(* Logix 5000 project; controller STAT 1756-L72 rev 20.12; software revision 20.04; part 14 of 34 *)
(* tags used below, declared in another part *)
   B14 : DINT[30];
   B15 : DINT[30];
   B16 : DINT[30];
   B17 : DINT[30];
   B3 : DINT[256];
   B9 : DINT[40];
   DateTime : DINT[7];   // DINT array tag for retrieve wallclock time through GSV created during conversion
   I19_000_Bit01 : ALIAS FOR I19[0].1;   // VANNE ALIBERT FERMEE
   I19_000_Bit07 : ALIAS FOR I19[0].7;   // LACK DETECTIE H2SO4
   I19_000_Bit08 : ALIAS FOR I19[0].8;   // LACK DETECTIE NAOH
   I19_001_Bit02 : ALIAS FOR I19[1].2;
   I19_001_Bit04 : ALIAS FOR I19[1].4;
   I1_008_Bit00 : ALIAS FOR I1[8].0;   // Noodstop gedrukt
   I1_008_Bit12 : ALIAS FOR I1[8].12;   // start
   I1_009_Bit00 : ALIAS FOR I1[9].0;   // Spanning 220 V nuts ok
   I1_009_Bit01 : ALIAS FOR I1[9].1;   // Spanning 220 v ac ok
   I1_009_Bit02 : ALIAS FOR I1[9].2;   // Spanning 24 v dc ok
   I1_009_Bit03 : ALIAS FOR I1[9].3;   // Thermische storing pomp 1
   I1_009_Bit07 : ALIAS FOR I1[9].7;   // Thermische storing pomp 2
   I1_009_Bit11 : ALIAS FOR I1[9].11;   // Thermische storing pomp 3
   I1_009_Bit15 : ALIAS FOR I1[9].15;   // Thermische storing pomp pd1 ok
   I1_010_Bit00 : ALIAS FOR I1[10].0;   // PD1 spanning ok op regelaar
   I1_010_Bit02 : ALIAS FOR I1[10].2;   // Thermische storng pomp pd2 ok
   I1_010_Bit03 : ALIAS FOR I1[10].3;   // PD2 spanning ok op regelaar
   I1_010_Bit05 : ALIAS FOR I1[10].5;   // Vlotterschak lal stormbekken
   I1_010_Bit06 : ALIAS FOR I1[10].6;   // Storing voeding promag 33
   I1_010_Bit08 : ALIAS FOR I1[10].8;   // Fout promag 33
   I1_010_Bit10 : ALIAS FOR I1[10].10;   // Noodstop relais ok stormbekken
   I1_016_Bit00 : ALIAS FOR I1[16].0;   // CL2 noodstop gedrukt
   I1_016_Bit10 : ALIAS FOR I1[16].10;   // conduc 3 alarm
   I1_016_Bit13 : ALIAS FOR I1[16].13;   // Niveau lus5 kontakt3
   I1_017_Bit00 : ALIAS FOR I1[17].0;   // CL3 noodstop gedrukt
   I1_017_Bit10 : ALIAS FOR I1[17].10;   // conduc 4 alarm
   I1_017_Bit13 : ALIAS FOR I1[17].13;   // Niveau lus6 kontakt3
   I1_017_Bit14 : ALIAS FOR I1[17].14;   // Niveau A3 vlotter niveau
   I1_018_Bit00 : ALIAS FOR I1[18].0;   // CL4 noodstop gedrukt
   I1_018_Bit10 : ALIAS FOR I1[18].10;   // conduc 5 alarm
   I1_018_Bit13 : ALIAS FOR I1[18].13;   // Niveau lus7 kontakt3
   I1_019_Bit00 : ALIAS FOR I1[19].0;   // 220V ok aan lijn 123
   I2_000_Bit00 : ALIAS FOR I2[0].0;   // Deelnoodstop cl2 lijn 1
   I2_000_Bit01 : ALIAS FOR I2[0].1;   // Deelnoodstop cl3 lijn 3
   I2_000_Bit02 : ALIAS FOR I2[0].2;   // Deelnoodstop cl4
   I2_000_Bit03 : ALIAS FOR I2[0].3;   // Deelnoodstop cl5 lijn 4
   I2_000_Bit04 : ALIAS FOR I2[0].4;   // Deelnoodstop cl6 eurowater
   I2_000_Bit05 : ALIAS FOR I2[0].5;   // Deelnoodstop cl7 IBT A
   I2_000_Bit06 : ALIAS FOR I2[0].6;   // Deelnoodstop cl7 IBT B
   I2_000_Bit07 : ALIAS FOR I2[0].7;   // Deelnoodstop cl7 IBT C
   I2_000_Bit08 : ALIAS FOR I2[0].8;   // Voeidng 220V ok
   I2_000_Bit09 : ALIAS FOR I2[0].9;   // Storing voeding lijn 1 cl 2
   I2_000_Bit10 : ALIAS FOR I2[0].10;   // Storing voeding lijn 2 cl 3
   I2_000_Bit11 : ALIAS FOR I2[0].11;   // Storing voeding lijn 3 cl 4
   I2_000_Bit12 : ALIAS FOR I2[0].12;   // Storing voeding lijn 4 cl 5
   I2_000_Bit13 : ALIAS FOR I2[0].13;   // Storing voeding lijn deel eurowater cl 6
   I2_000_Bit14 : ALIAS FOR I2[0].14;   // Storing voedingslijn IBT-A CL 7
   I2_000_Bit15 : ALIAS FOR I2[0].15;   // Storing voedingslijn IBT-B CL 8
   I2_001_Bit00 : ALIAS FOR I2[1].0;   // Storing voedingslijn IBT-C CL 9
   I2_001_Bit01 : ALIAS FOR I2[1].1;   // Voeding meting 220V ok
   I2_001_Bit02 : ALIAS FOR I2[1].2;   // Voeding DC 24 ok
   I2_001_Bit03 : ALIAS FOR I2[1].3;   // Storing voeding 24V DC algemeen
   I2_001_Bit04 : ALIAS FOR I2[1].4;   // Storing voeding 24V ingangen
   I2_001_Bit05 : ALIAS FOR I2[1].5;   // Storing 24V meting
   I2_001_Bit06 : ALIAS FOR I2[1].6;   // Voeding uitgang 24V
   I2_001_Bit08 : ALIAS FOR I2[1].8;   // Motor p11 lijn1 thermische storing
   I2_001_Bit10 : ALIAS FOR I2[1].10;   // Motor p12 lijn1 thermische storing
   I2_001_Bit12 : ALIAS FOR I2[1].12;   // Motor p13 lijn2 thermische storing
   I2_001_Bit14 : ALIAS FOR I2[1].14;   // Motor p14 lijn2 thermische storing
   I3_000_Bit00 : ALIAS FOR I3[0].0;   // Motor p15 lijn3 thermische storing
   I3_000_Bit02 : ALIAS FOR I3[0].2;   // Motor p16 lijn3 thermische storing
   I3_000_Bit04 : ALIAS FOR I3[0].4;   // Motor p17 lijn4 thermische storing
   I3_000_Bit06 : ALIAS FOR I3[0].6;   // Motor p18 lijn4 thermische storing
   I3_000_Bit07 : ALIAS FOR I3[0].7;   // Motor pro 1 voedingpomp osmose 1 Thermische storing
   I3_000_Bit09 : ALIAS FOR I3[0].9;   // Motor pro 1 voedingpomp osmose 1 in driehoek
   I3_000_Bit11 : ALIAS FOR I3[0].11;   // Motor pro2 voedingpomp osmose 2 Thermische storing
   I3_000_Bit13 : ALIAS FOR I3[0].13;   // Motor pro 2 voedingpomp osmose 2 in driehoek
   I3_000_Bit15 : ALIAS FOR I3[0].15;   // Motor P21 Thermische storing Kuip AZ
   I3_001_Bit03 : ALIAS FOR I3[1].3;   // Thermische storing motor P22 kuip AZ
   I3_001_Bit07 : ALIAS FOR I3[1].7;   // Thermische storing motor PRO3 voedingsp. osmose 3
   I3_001_Bit09 : ALIAS FOR I3[1].9;   // Motor voedingspomp osmose 3 in drie
   I3_001_Bit11 : ALIAS FOR I3[1].11;   // Motor P21 reinigingspomp membraam
   I3_001_Bit13 : ALIAS FOR I3[1].13;   // Thermische storing S2 ventilator
   I3_001_Bit15 : ALIAS FOR I3[1].15;   // Thermische storing voedingspomp fabriek 1
   I4_000_Bit03 : ALIAS FOR I4[0].3;   // Thermische storing voedingspomp fabriek 2
   I4_000_Bit08 : ALIAS FOR I4[0].8;   // Thermische storing motor p 5 ok
   I4_000_Bit10 : ALIAS FOR I4[0].10;   // Thermische storing p6 ok
   I4_000_Bit15 : ALIAS FOR I4[0].15;   // thermische storing frequentieregelaar motor p25
   I4_001_Bit01 : ALIAS FOR I4[1].1;   // Thermische storing freqreg p20
   I4_001_Bit03 : ALIAS FOR I4[1].3;   // Motor AG1 mixer vat neutral thermische st ok
   I4_001_Bit05 : ALIAS FOR I4[1].5;   // Motor acide thermische st ok
   I4_001_Bit07 : ALIAS FOR I4[1].7;   // Motor acide 4 thermische st ok
   I4_001_Bit09 : ALIAS FOR I4[1].9;   // Motor soude 5 thermische st ok
   I4_001_Bit11 : ALIAS FOR I4[1].11;   // Motor soude 6 thermische st ok
   I4_001_Bit13 : ALIAS FOR I4[1].13;   // Motor ag2 mixer thermische st ok
   I4_001_Bit15 : ALIAS FOR I4[1].15;   // Motor ag3 mixer thermische st ok
   I5_000_Bit00 : ALIAS FOR I5[0].0;   // thermische storing motor doseerpop1 pd7
   I5_000_Bit01 : ALIAS FOR I5[0].1;   // spanning op motor freqreg doseer floculaat
   I5_000_Bit02 : ALIAS FOR I5[0].2;   // storing freqreg doseer floculaat
   I5_000_Bit03 : ALIAS FOR I5[0].3;   // thermische storing motor freqreg doseer floculaat pd8
   I5_000_Bit04 : ALIAS FOR I5[0].4;   // spanning op motor freqreg doseer floculaat pd8
   I5_000_Bit05 : ALIAS FOR I5[0].5;   // storing freqreg doseer floculaat pd8
   I5_000_Bit07 : ALIAS FOR I5[0].7;   // thermische storing motor zuiveringspomp p19
   I5_000_Bit09 : ALIAS FOR I5[0].9;   // thermische storing motor zuiveringspomp p19b
   I5_000_Bit10 : ALIAS FOR I5[0].10;   // thermische storing motor PM1
   I5_000_Bit11 : ALIAS FOR I5[0].11;   // spanning op motor freqreg recerculatiep. dec. ingang 1
   I5_000_Bit12 : ALIAS FOR I5[0].12;   // fout freqreg recerculatiep. dec. ingang 1
   I5_000_Bit13 : ALIAS FOR I5[0].13;   // thermische storing motor recirculatiep. dec. ingang 2
   I5_000_Bit14 : ALIAS FOR I5[0].14;   // spanning freqreg. recirculatiep. dec. ingang 2
   I5_000_Bit15 : ALIAS FOR I5[0].15;   // fout freqreg recerculatiep. dec. ingang 2
   I5_001_Bit00 : ALIAS FOR I5[1].0;   // thermische storing motor evacuatiepomp dec. ingang 1
   I5_001_Bit01 : ALIAS FOR I5[1].1;   // spanning freqreg. evacuatiepomp decanter ingang 1
   I5_001_Bit02 : ALIAS FOR I5[1].2;   // fout freqreg pm3 evacuatiep. dec. ingang 1
   I5_001_Bit03 : ALIAS FOR I5[1].3;   // thermische storing motor evacuatiepomp dec. ingang 2
   I5_001_Bit04 : ALIAS FOR I5[1].4;   // spanning freqreg. evacuatiepomp decanter ingang 2
   I5_001_Bit05 : ALIAS FOR I5[1].5;   // fout freqreg pm4 evacuatiep. dec. ingang 2
   I5_001_Bit06 : ALIAS FOR I5[1].6;   // thermische storing voedingspomp 1 osmose ok
   I5_001_Bit08 : ALIAS FOR I5[1].8;   // thermische storing voedingspomp 2 osmose ok
   I5_001_Bit10 : ALIAS FOR I5[1].10;   // thermische storing voedingspomp 3 osmose ok
   I6_000_Bit10 : ALIAS FOR I6[0].10;   // pressostaat osmose1
   I6_000_Bit11 : ALIAS FOR I6[0].11;   // pressostaat osmose2
   I6_000_Bit12 : ALIAS FOR I6[0].12;   // pressostaat osmose3
   I6_001_Bit06 : ALIAS FOR I6[1].6;   // debietsmeting q2 fout 1
   I6_001_Bit09 : ALIAS FOR I6[1].9;   // debietsmeting q3 fout 1
   I6_001_Bit11 : ALIAS FOR I6[1].11;   // Ph meting vervuild water kontakt 1
   I7_000_Bit00 : ALIAS FOR I7[0].0;   // ph meting fout gerecycleerd water
   I7_000_Bit01 : ALIAS FOR I7[0].1;   // lus2 niveau kontakt 1
   I7_000_Bit03 : ALIAS FOR I7[0].3;   // lus2 niveau kontakt 3
   I7_000_Bit04 : ALIAS FOR I7[0].4;   // lus3 niveau kontakt 1
   I7_000_Bit06 : ALIAS FOR I7[0].6;   // lus3 niveau kontakt 3
   I7_000_Bit10 : ALIAS FOR I7[0].10;   // zeer hoog alarm ketel clarifee
   I7_000_Bit13 : ALIAS FOR I7[0].13;   // zeer laag alarm ketel clarifee
   I7_001_Bit03 : ALIAS FOR I7[1].3;   // Conductiviteit 1 alarm 3
   I7_001_Bit06 : ALIAS FOR I7[1].6;   // Conductiviteit 2 kontakt alarm
   I7_001_Bit12 : ALIAS FOR I7[1].12;   // Lus 8 niveau kontakt 3
   N12 : DINT[230];
   N13 : DINT[230];
   N26 : DINT[256];
   O14_001_Bit13 : ALIAS FOR O14[1].13;   // RO1_EV2 RO1_EV2
   O15_000_Bit01 : ALIAS FOR O15[0].1;   // RO2_EV2 RO2_EV2
   O15_000_Bit05 : ALIAS FOR O15[0].5;   // RO3_EV2 RO3_EV2
   O1_011_Bit00 : ALIAS FOR O1[11].0;
   O1_011_Bit03 : ALIAS FOR O1[11].3;
   T27 : TIMER[100];
   T4 : TIMER[200];
(* ibt, continued *)

ROUTINE _17_DEF_TEL   (* ladder *)
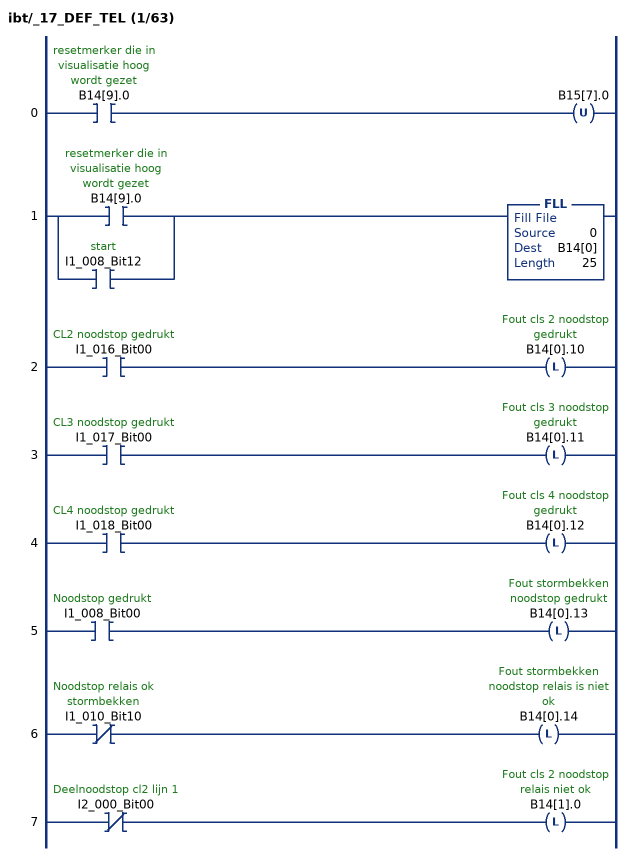
   0: XIC(B14[9].0)OTU(B15[7].0);
   1: [XIC(B14[9].0) ,XIC(I1_008_Bit12) ]FLL(0,B14[0],25);
   2: XIC(I1_016_Bit00)OTL(B14[0].10);
   3: XIC(I1_017_Bit00)OTL(B14[0].11);
   4: XIC(I1_018_Bit00)OTL(B14[0].12);
   5: XIC(I1_008_Bit00)OTL(B14[0].13);
   6: XIO(I1_010_Bit10)OTL(B14[0].14);
   7: XIO(I2_000_Bit00)OTL(B14[1].0);
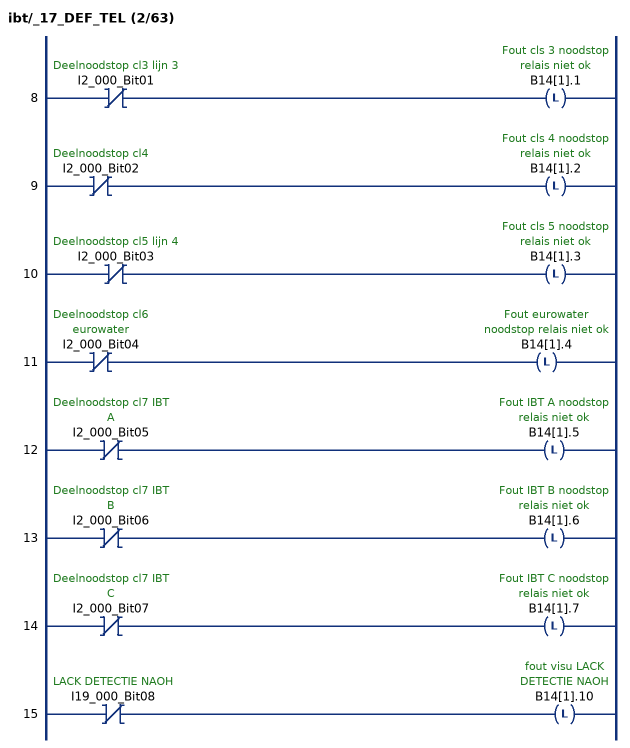
   8: XIO(I2_000_Bit01)OTL(B14[1].1);
   9: XIO(I2_000_Bit02)OTL(B14[1].2);
   10: XIO(I2_000_Bit03)OTL(B14[1].3);
   11: XIO(I2_000_Bit04)OTL(B14[1].4);
   12: XIO(I2_000_Bit05)OTL(B14[1].5);
   13: XIO(I2_000_Bit06)OTL(B14[1].6);
   14: XIO(I2_000_Bit07)OTL(B14[1].7);
   15: XIO(I19_000_Bit08)OTL(B14[1].10);
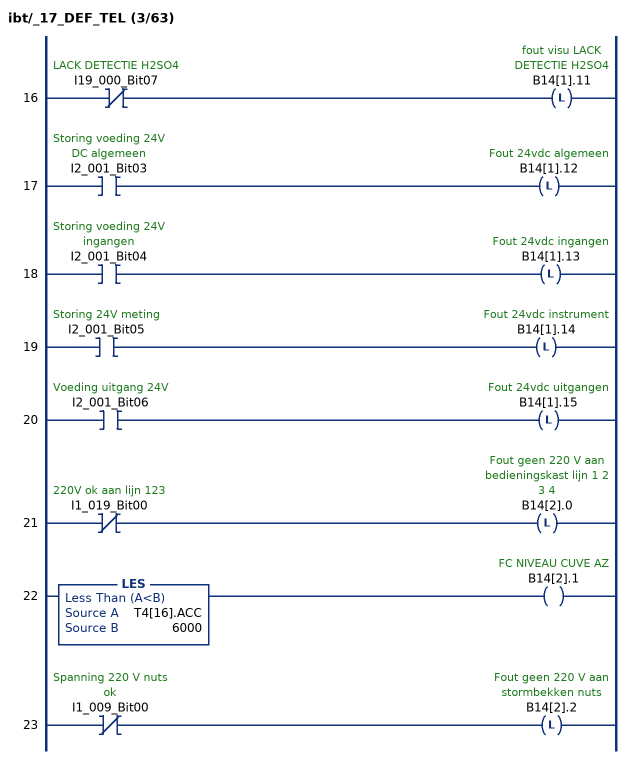
   16: XIO(I19_000_Bit07)OTL(B14[1].11);
   17: XIC(I2_001_Bit03)OTL(B14[1].12);
   18: XIC(I2_001_Bit04)OTL(B14[1].13);
   19: XIC(I2_001_Bit05)OTL(B14[1].14);
   20: XIC(I2_001_Bit06)OTL(B14[1].15);
   21: XIO(I1_019_Bit00)OTL(B14[2].0);
   22: LES(T4[16].ACC,6000)OTE(B14[2].1);
   23: XIO(I1_009_Bit00)OTL(B14[2].2);
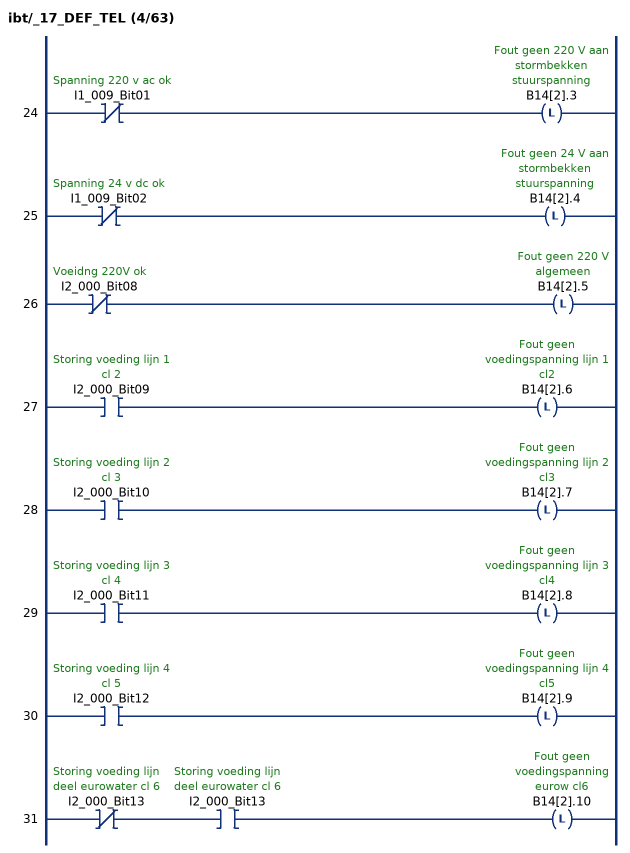
   24: XIO(I1_009_Bit01)OTL(B14[2].3);
   25: XIO(I1_009_Bit02)OTL(B14[2].4);
   26: XIO(I2_000_Bit08)OTL(B14[2].5);
   27: XIC(I2_000_Bit09)OTL(B14[2].6);
   28: XIC(I2_000_Bit10)OTL(B14[2].7);
   29: XIC(I2_000_Bit11)OTL(B14[2].8);
   30: XIC(I2_000_Bit12)OTL(B14[2].9);
   31: XIO(I2_000_Bit13)XIC(I2_000_Bit13)OTL(B14[2].10);
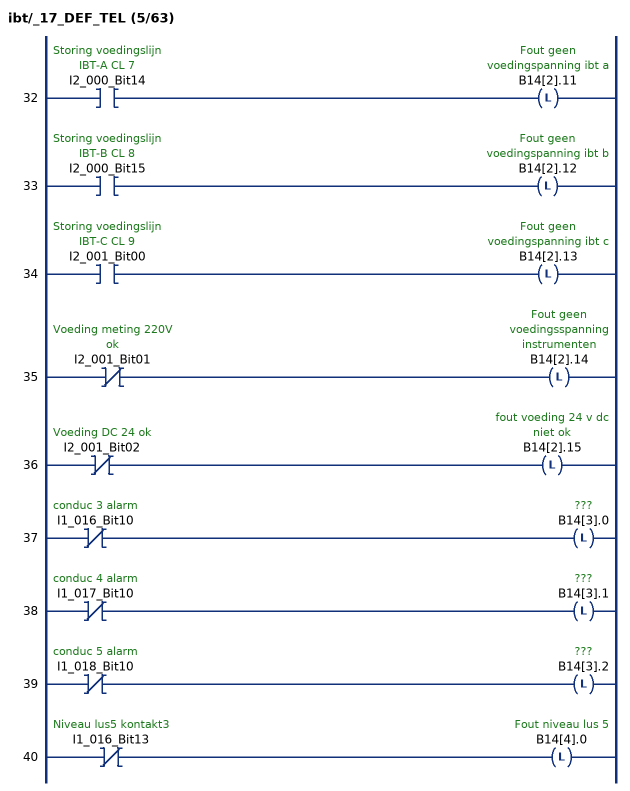
   32: XIC(I2_000_Bit14)OTL(B14[2].11);
   33: XIC(I2_000_Bit15)OTL(B14[2].12);
   34: XIC(I2_001_Bit00)OTL(B14[2].13);
   35: XIO(I2_001_Bit01)OTL(B14[2].14);
   36: XIO(I2_001_Bit02)OTL(B14[2].15);
   37: XIO(I1_016_Bit10)OTL(B14[3].0);
   38: XIO(I1_017_Bit10)OTL(B14[3].1);
   39: XIO(I1_018_Bit10)OTL(B14[3].2);
   40: XIO(I1_016_Bit13)OTL(B14[4].0);
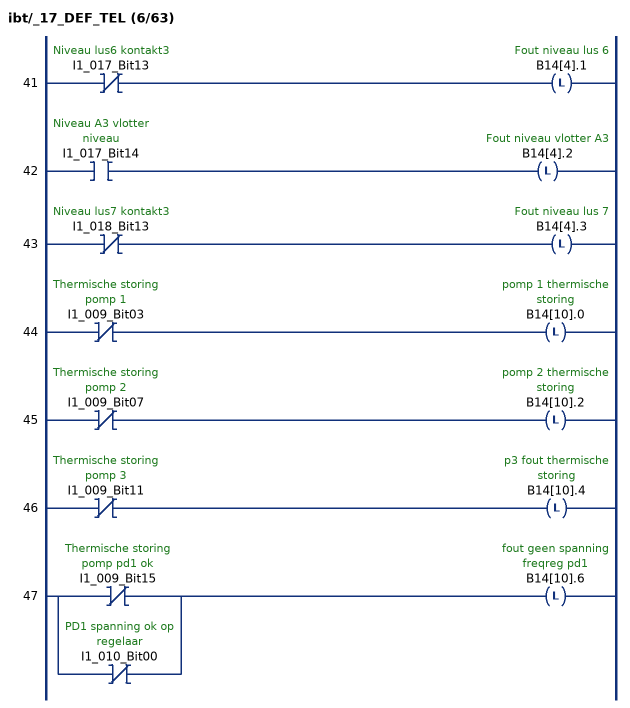
   41: XIO(I1_017_Bit13)OTL(B14[4].1);
   42: XIC(I1_017_Bit14)OTL(B14[4].2);
   43: XIO(I1_018_Bit13)OTL(B14[4].3);
   44: XIO(I1_009_Bit03)OTL(B14[10].0);
   45: XIO(I1_009_Bit07)OTL(B14[10].2);
   46: XIO(I1_009_Bit11)OTL(B14[10].4);
   47: [XIO(I1_009_Bit15) ,XIO(I1_010_Bit00) ]OTL(B14[10].6);
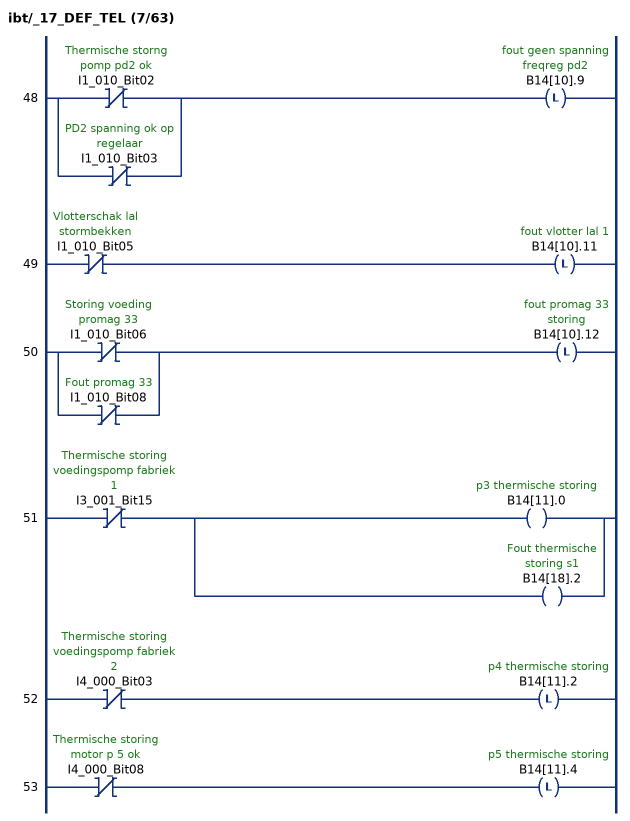
   48: [XIO(I1_010_Bit02) ,XIO(I1_010_Bit03) ]OTL(B14[10].9);
   49: XIO(I1_010_Bit05)OTL(B14[10].11);
   50: [XIO(I1_010_Bit06) ,XIO(I1_010_Bit08) ]OTL(B14[10].12);
   51: XIO(I3_001_Bit15)[OTE(B14[11].0) ,OTE(B14[18].2) ];
   52: XIO(I4_000_Bit03)OTL(B14[11].2);
   53: XIO(I4_000_Bit08)OTL(B14[11].4);
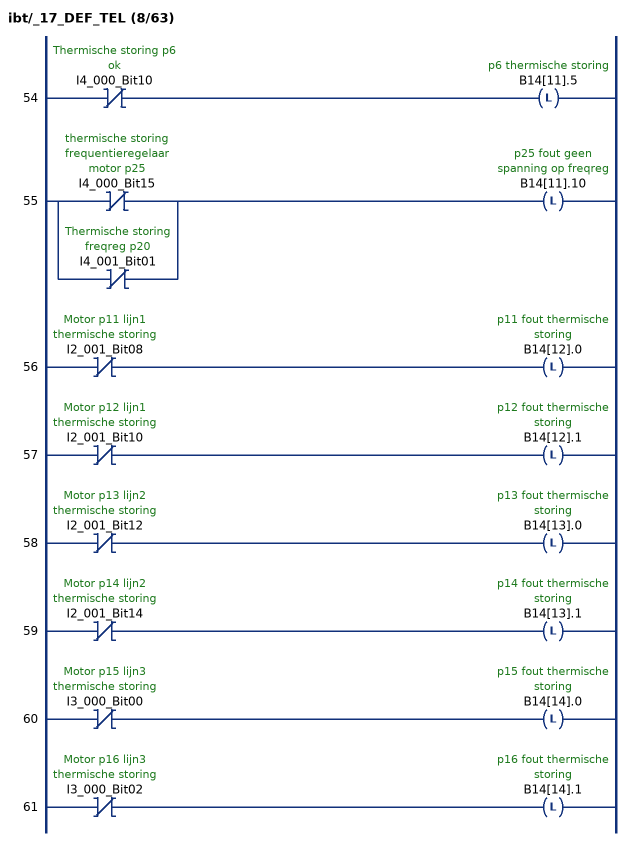
   54: XIO(I4_000_Bit10)OTL(B14[11].5);
   55: [XIO(I4_000_Bit15) ,XIO(I4_001_Bit01) ]OTL(B14[11].10);
   56: XIO(I2_001_Bit08)OTL(B14[12].0);
   57: XIO(I2_001_Bit10)OTL(B14[12].1);
   58: XIO(I2_001_Bit12)OTL(B14[13].0);
   59: XIO(I2_001_Bit14)OTL(B14[13].1);
   60: XIO(I3_000_Bit00)OTL(B14[14].0);
   61: XIO(I3_000_Bit02)OTL(B14[14].1);
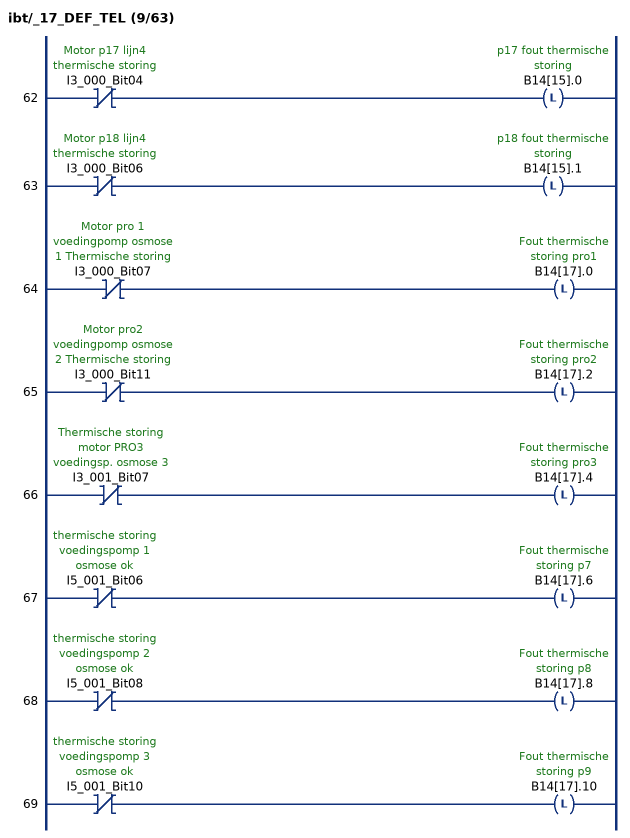
   62: XIO(I3_000_Bit04)OTL(B14[15].0);
   63: XIO(I3_000_Bit06)OTL(B14[15].1);
   64: XIO(I3_000_Bit07)OTL(B14[17].0);
   65: XIO(I3_000_Bit11)OTL(B14[17].2);
   66: XIO(I3_001_Bit07)OTL(B14[17].4);
   67: XIO(I5_001_Bit06)OTL(B14[17].6);
   68: XIO(I5_001_Bit08)OTL(B14[17].8);
   69: XIO(I5_001_Bit10)OTL(B14[17].10);
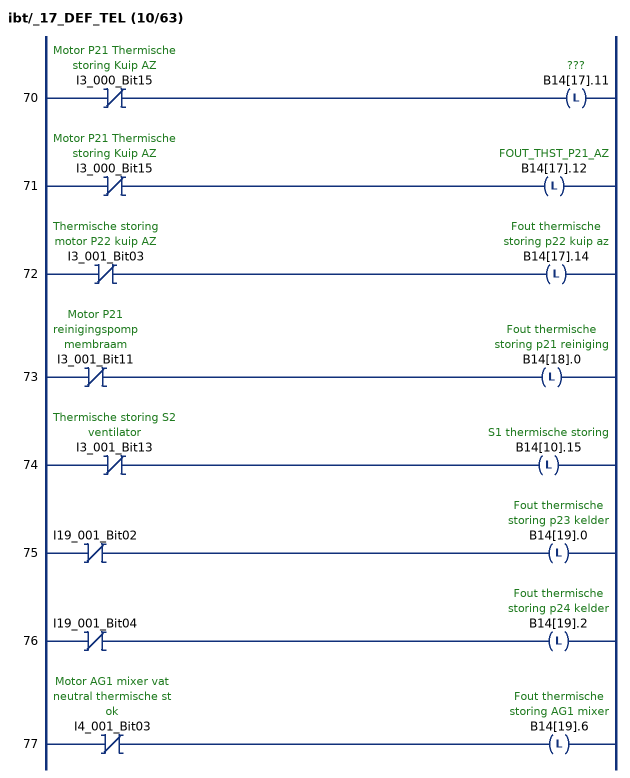
   70: XIO(I3_000_Bit15)OTL(B14[17].11);
   71: XIO(I3_000_Bit15)OTL(B14[17].12);
   72: XIO(I3_001_Bit03)OTL(B14[17].14);
   73: XIO(I3_001_Bit11)OTL(B14[18].0);
   74: XIO(I3_001_Bit13)OTL(B14[10].15);
   75: XIO(I19_001_Bit02)OTL(B14[19].0);
   76: XIO(I19_001_Bit04)OTL(B14[19].2);
   77: XIO(I4_001_Bit03)OTL(B14[19].6);
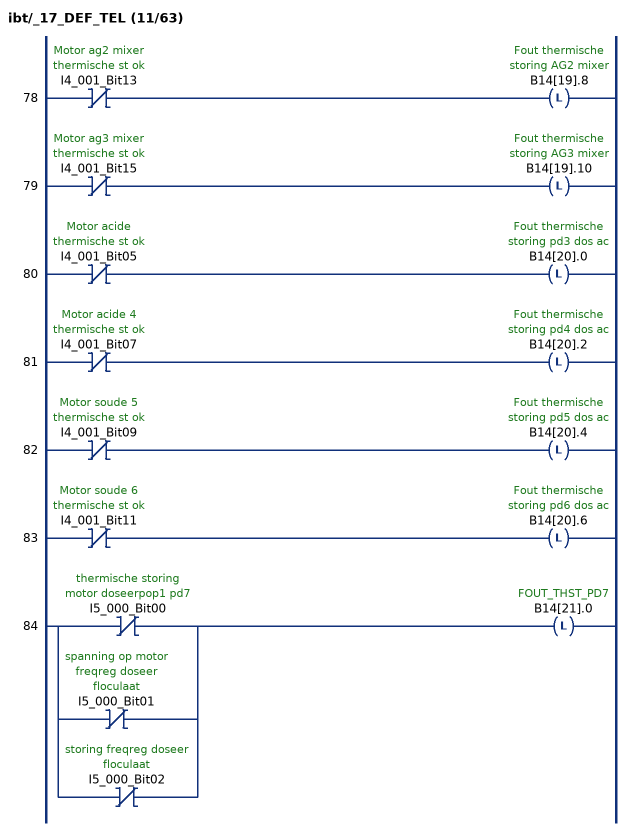
   78: XIO(I4_001_Bit13)OTL(B14[19].8);
   79: XIO(I4_001_Bit15)OTL(B14[19].10);
   80: XIO(I4_001_Bit05)OTL(B14[20].0);
   81: XIO(I4_001_Bit07)OTL(B14[20].2);
   82: XIO(I4_001_Bit09)OTL(B14[20].4);
   83: XIO(I4_001_Bit11)OTL(B14[20].6);
   84: [XIO(I5_000_Bit00) ,[XIO(I5_000_Bit01) ,XIO(I5_000_Bit02) ] ]OTL(B14[21].0);
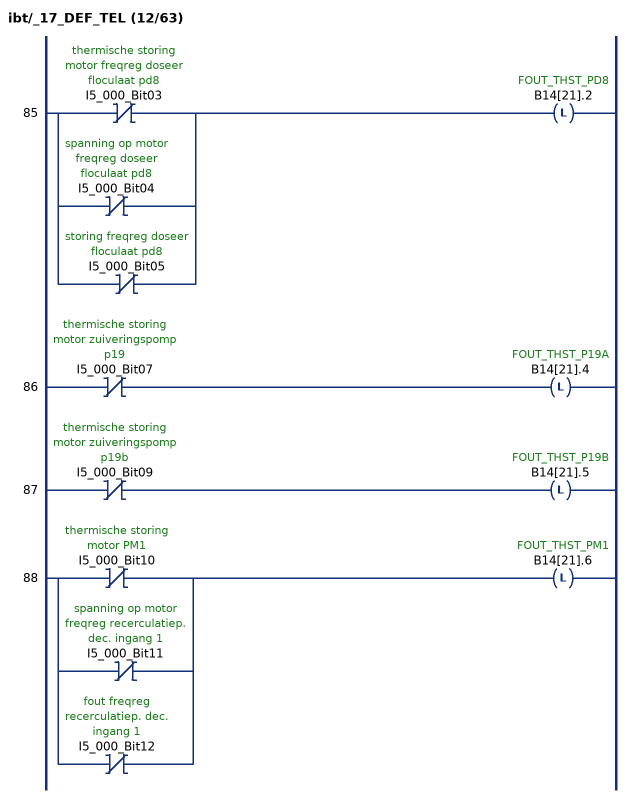
   85: [XIO(I5_000_Bit03) ,[XIO(I5_000_Bit04) ,XIO(I5_000_Bit05) ] ]OTL(B14[21].2);
   86: XIO(I5_000_Bit07)OTL(B14[21].4);
   87: XIO(I5_000_Bit09)OTL(B14[21].5);
   88: [XIO(I5_000_Bit10) ,[XIO(I5_000_Bit11) ,XIO(I5_000_Bit12) ] ]OTL(B14[21].6);
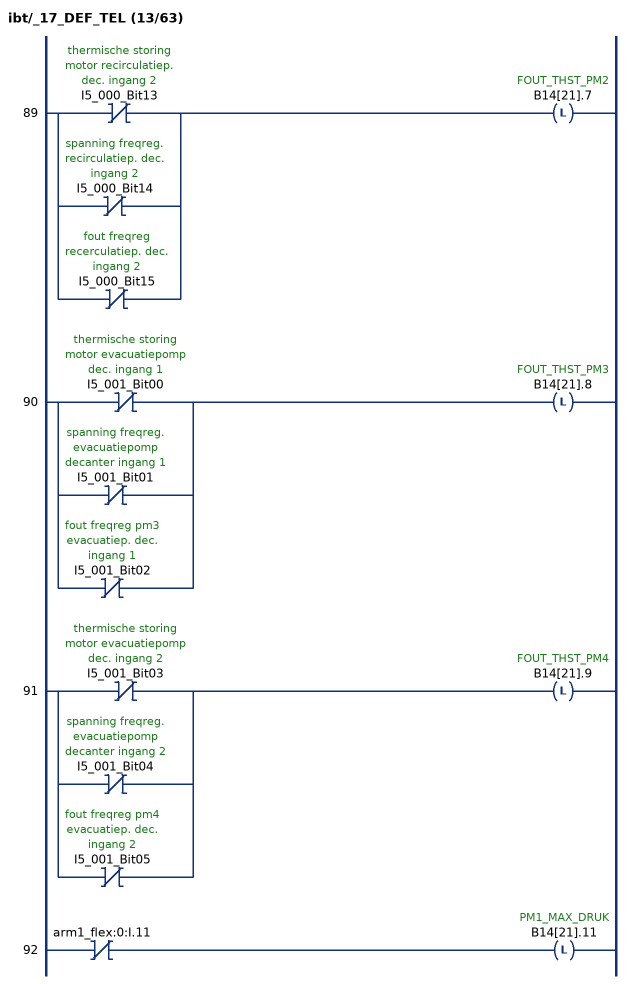
   89: [XIO(I5_000_Bit13) ,[XIO(I5_000_Bit14) ,XIO(I5_000_Bit15) ] ]OTL(B14[21].7);
   90: [XIO(I5_001_Bit00) ,[XIO(I5_001_Bit01) ,XIO(I5_001_Bit02) ] ]OTL(B14[21].8);
   91: [XIO(I5_001_Bit03) ,[XIO(I5_001_Bit04) ,XIO(I5_001_Bit05) ] ]OTL(B14[21].9);
   92: XIO(arm1_flex:0:I.11)OTL(B14[21].11);
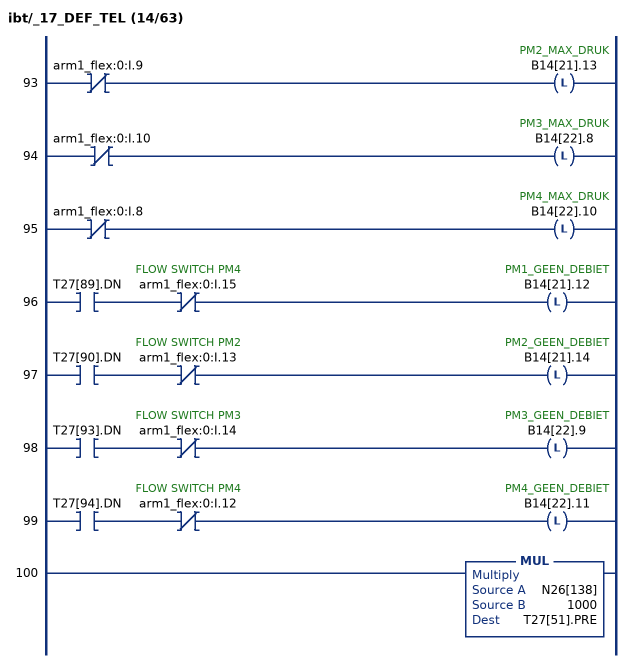
   93: XIO(arm1_flex:0:I.9)OTL(B14[21].13);
   94: XIO(arm1_flex:0:I.10)OTL(B14[22].8);
   95: XIO(arm1_flex:0:I.8)OTL(B14[22].10);
   96: XIC(T27[89].DN)XIO(arm1_flex:0:I.15)OTL(B14[21].12);
   97: XIC(T27[90].DN)XIO(arm1_flex:0:I.13)OTL(B14[21].14);
   98: XIC(T27[93].DN)XIO(arm1_flex:0:I.14)OTL(B14[22].9);
   99: XIC(T27[94].DN)XIO(arm1_flex:0:I.12)OTL(B14[22].11);
   100: MUL(N26[138],1000,T27[51].PRE);
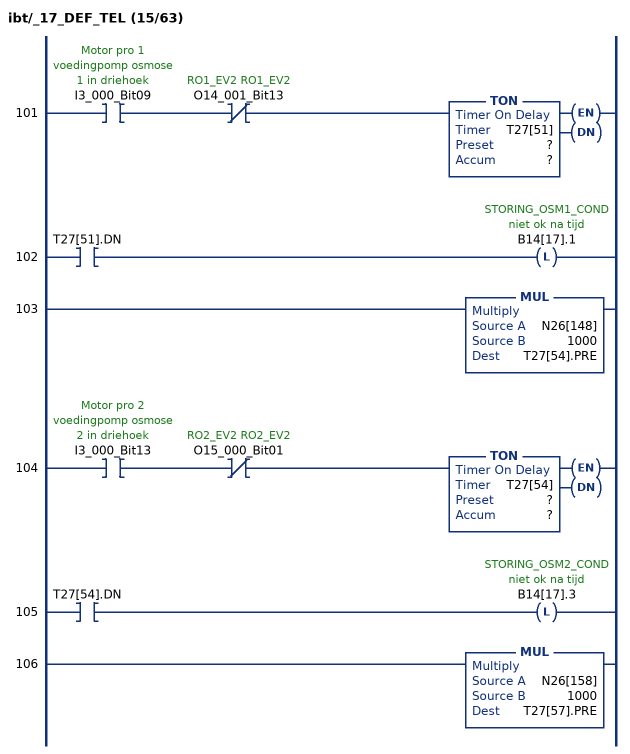
   101: XIC(I3_000_Bit09)XIO(O14_001_Bit13)TON(T27[51],?,?);
   102: XIC(T27[51].DN)OTL(B14[17].1);
   103: MUL(N26[148],1000,T27[54].PRE);
   104: XIC(I3_000_Bit13)XIO(O15_000_Bit01)TON(T27[54],?,?);
   105: XIC(T27[54].DN)OTL(B14[17].3);
   106: MUL(N26[158],1000,T27[57].PRE);
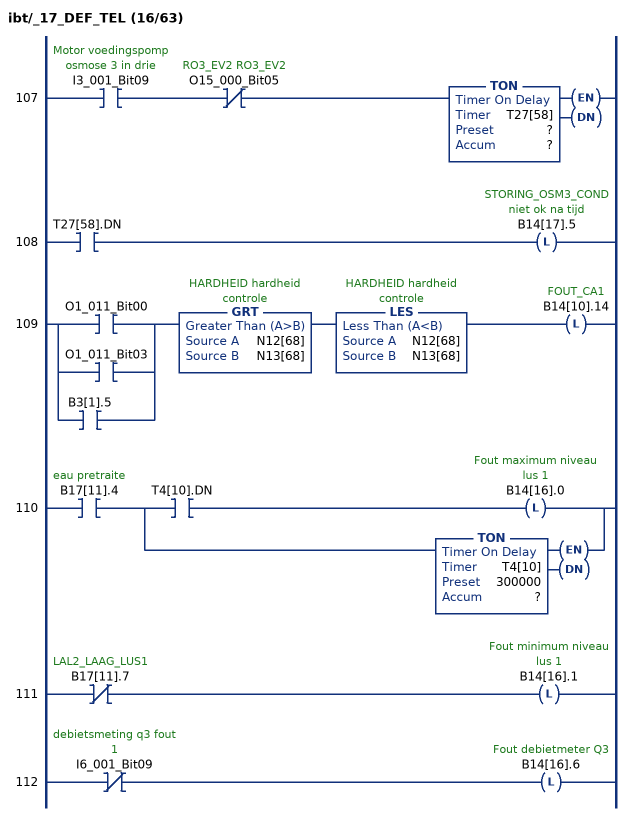
   107: XIC(I3_001_Bit09)XIO(O15_000_Bit05)TON(T27[58],?,?);
   108: XIC(T27[58].DN)OTL(B14[17].5);
   109: [XIC(O1_011_Bit00) ,XIC(O1_011_Bit03) ,XIC(B3[1].5) ]GRT(N12[68],N13[68])LES(N12[68],N13[68])OTL(B14[10].14);
   110: XIC(B17[11].4)[XIC(T4[10].DN) OTL(B14[16].0) ,TON(T4[10],?,?) ];
   111: XIO(B17[11].7)OTL(B14[16].1);
   112: XIO(I6_001_Bit09)OTL(B14[16].6);
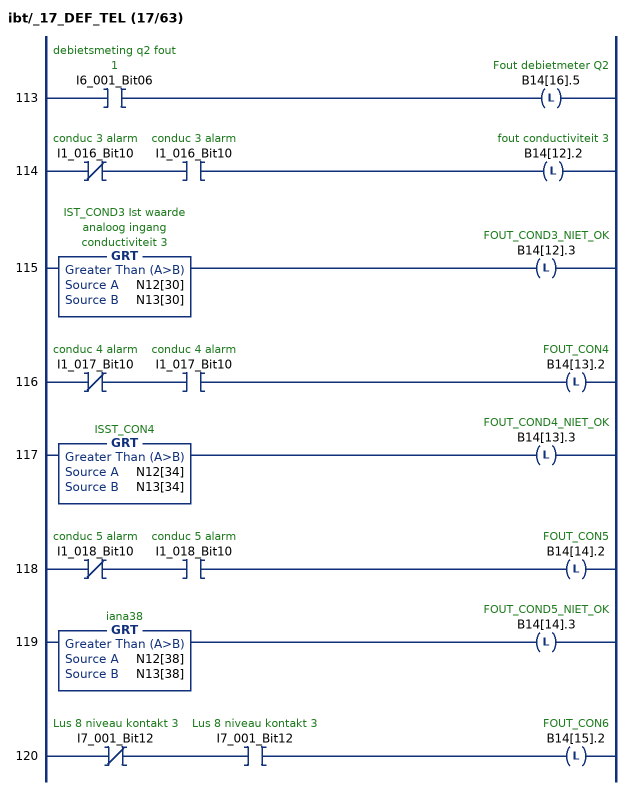
   113: XIC(I6_001_Bit06)OTL(B14[16].5);
   114: XIO(I1_016_Bit10)XIC(I1_016_Bit10)OTL(B14[12].2);
   115: GRT(N12[30],N13[30])OTL(B14[12].3);
   116: XIO(I1_017_Bit10)XIC(I1_017_Bit10)OTL(B14[13].2);
   117: GRT(N12[34],N13[34])OTL(B14[13].3);
   118: XIO(I1_018_Bit10)XIC(I1_018_Bit10)OTL(B14[14].2);
   119: GRT(N12[38],N13[38])OTL(B14[14].3);
   120: XIO(I7_001_Bit12)XIC(I7_001_Bit12)OTL(B14[15].2);
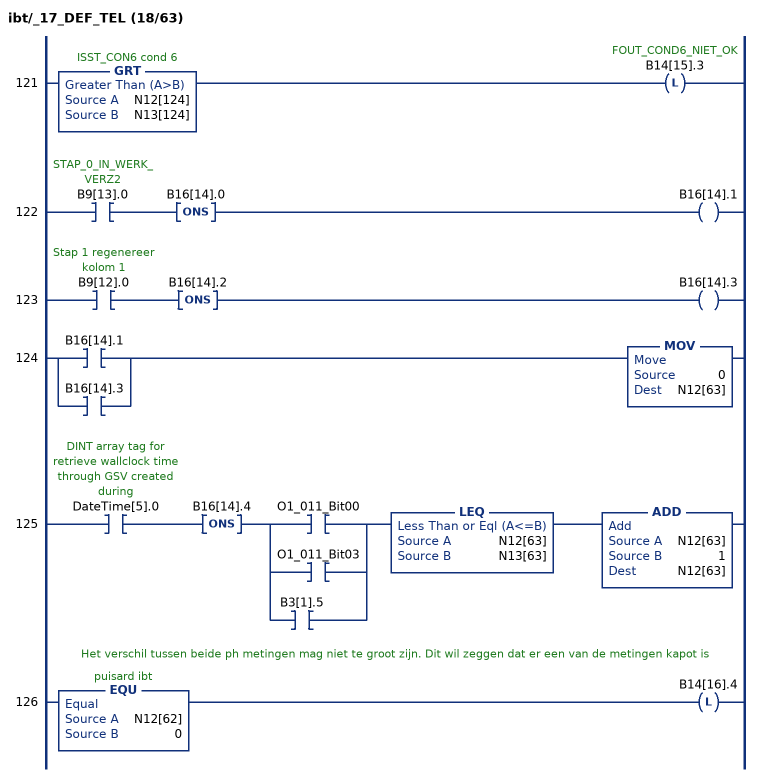
   121: GRT(N12[124],N13[124])OTL(B14[15].3);
   122: XIC(B9[13].0)ONS(B16[14].0)OTE(B16[14].1);
   123: XIC(B9[12].0)ONS(B16[14].2)OTE(B16[14].3);
   124: [XIC(B16[14].1) ,XIC(B16[14].3) ]MOV(0,N12[63]);
   125: XIC(DateTime[5].0)ONS(B16[14].4)[XIC(O1_011_Bit00) ,XIC(O1_011_Bit03) ,XIC(B3[1].5) ]LEQ(N12[63],N13[63])ADD(N12[63],1,N12[63]);
   // Het verschil tussen beide ph metingen mag niet te groot zijn. Dit wil zeggen dat er een van de metingen kapot is
   126: EQU(N12[62],0)OTL(B14[16].4);
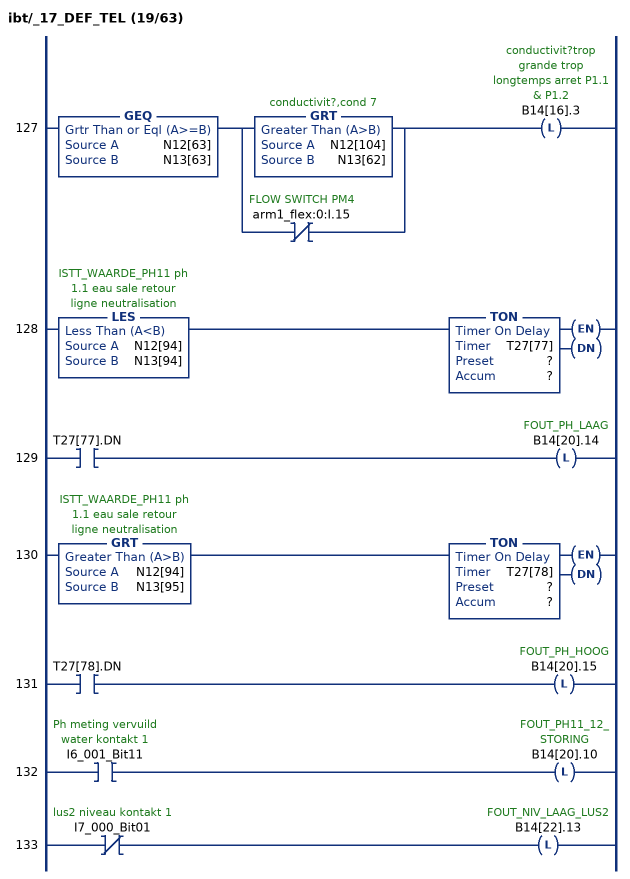
   127: GEQ(N12[63],N13[63])[GRT(N12[104],N13[62]) ,XIO(arm1_flex:0:I.15) ]OTL(B14[16].3);
   128: LES(N12[94],N13[94])TON(T27[77],?,?);
   129: XIC(T27[77].DN)OTL(B14[20].14);
   130: GRT(N12[94],N13[95])TON(T27[78],?,?);
   131: XIC(T27[78].DN)OTL(B14[20].15);
   132: XIC(I6_001_Bit11)OTL(B14[20].10);
   133: XIO(I7_000_Bit01)OTL(B14[22].13);
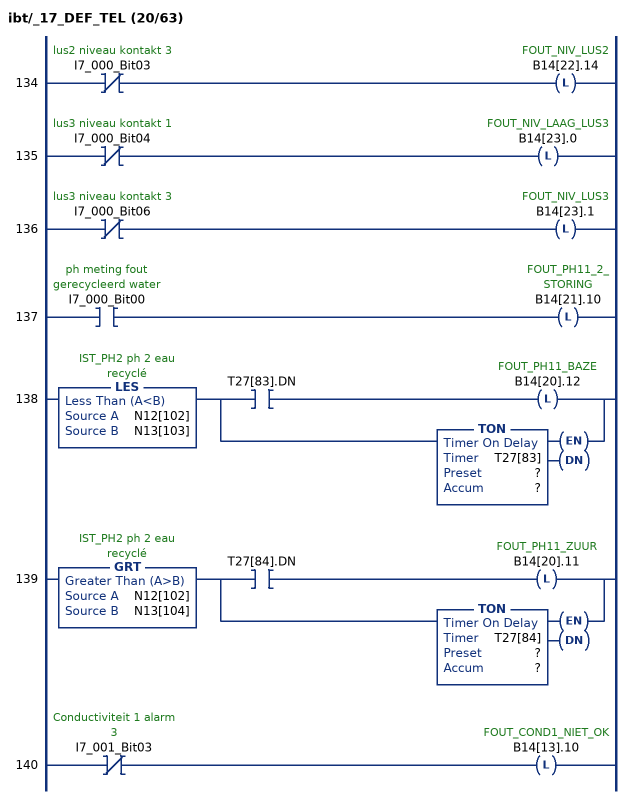
   134: XIO(I7_000_Bit03)OTL(B14[22].14);
   135: XIO(I7_000_Bit04)OTL(B14[23].0);
   136: XIO(I7_000_Bit06)OTL(B14[23].1);
   137: XIC(I7_000_Bit00)OTL(B14[21].10);
   138: LES(N12[102],N13[103])[XIC(T27[83].DN) OTL(B14[20].12) ,TON(T27[83],?,?) ];
   139: GRT(N12[102],N13[104])[XIC(T27[84].DN) OTL(B14[20].11) ,TON(T27[84],?,?) ];
   140: XIO(I7_001_Bit03)OTL(B14[13].10);
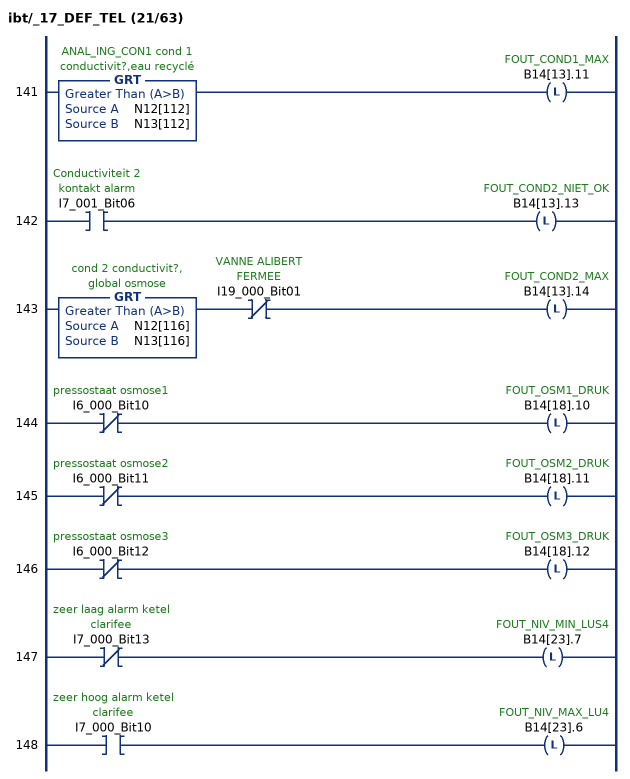
   141: GRT(N12[112],N13[112])OTL(B14[13].11);
   142: XIC(I7_001_Bit06)OTL(B14[13].13);
   143: GRT(N12[116],N13[116])XIO(I19_000_Bit01)OTL(B14[13].14);
   144: XIO(I6_000_Bit10)OTL(B14[18].10);
   145: XIO(I6_000_Bit11)OTL(B14[18].11);
   146: XIO(I6_000_Bit12)OTL(B14[18].12);
   147: XIO(I7_000_Bit13)OTL(B14[23].7);
   148: XIC(I7_000_Bit10)OTL(B14[23].6);
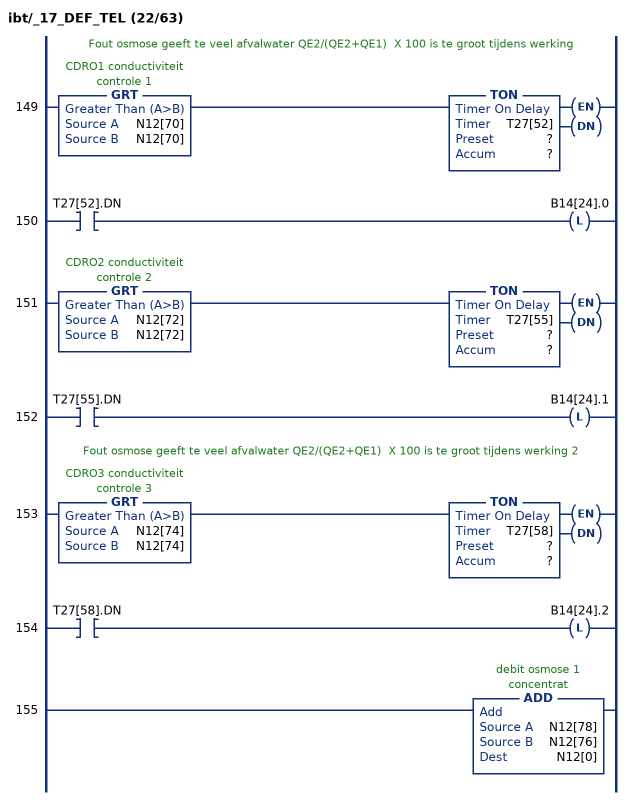
   // Fout osmose geeft te veel afvalwater QE2/(QE2+QE1)  X 100 is te groot tijdens werking
   149: GRT(N12[70],N12[70])TON(T27[52],?,?);
   150: XIC(T27[52].DN)OTL(B14[24].0);
   151: GRT(N12[72],N12[72])TON(T27[55],?,?);
   152: XIC(T27[55].DN)OTL(B14[24].1);
   // Fout osmose geeft te veel afvalwater QE2/(QE2+QE1)  X 100 is te groot tijdens werking 2
   153: GRT(N12[74],N12[74])TON(T27[58],?,?);
   154: XIC(T27[58].DN)OTL(B14[24].2);
   155: ADD(N12[78],N12[76],N12[0]);
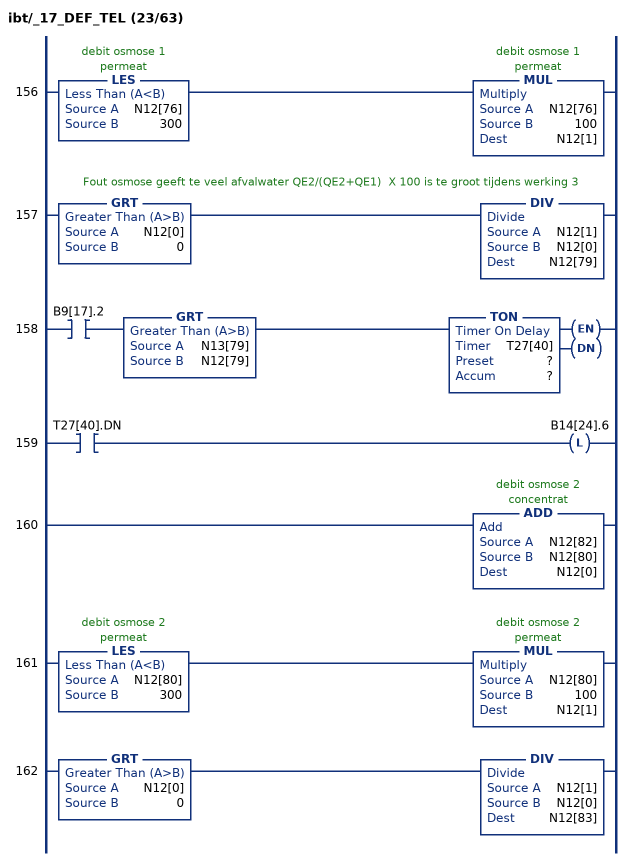
   156: LES(N12[76],300)MUL(N12[76],100,N12[1]);
   // Fout osmose geeft te veel afvalwater QE2/(QE2+QE1)  X 100 is te groot tijdens werking 3
   157: GRT(N12[0],0)DIV(N12[1],N12[0],N12[79]);
   158: XIC(B9[17].2)GRT(N13[79],N12[79])TON(T27[40],?,?);
   159: XIC(T27[40].DN)OTL(B14[24].6);
   160: ADD(N12[82],N12[80],N12[0]);
   161: LES(N12[80],300)MUL(N12[80],100,N12[1]);
   162: GRT(N12[0],0)DIV(N12[1],N12[0],N12[83]);
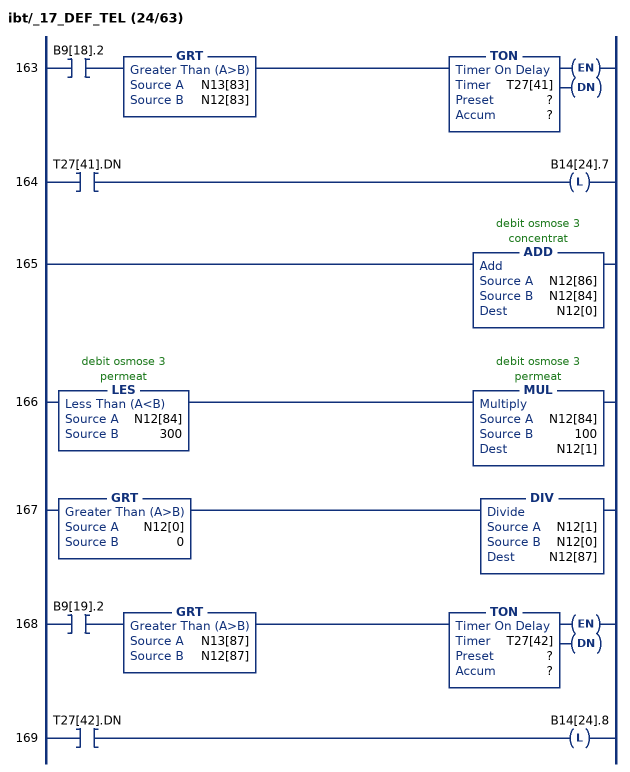
   163: XIC(B9[18].2)GRT(N13[83],N12[83])TON(T27[41],?,?);
   164: XIC(T27[41].DN)OTL(B14[24].7);
   165: ADD(N12[86],N12[84],N12[0]);
   166: LES(N12[84],300)MUL(N12[84],100,N12[1]);
   167: GRT(N12[0],0)DIV(N12[1],N12[0],N12[87]);
   168: XIC(B9[19].2)GRT(N13[87],N12[87])TON(T27[42],?,?);
   169: XIC(T27[42].DN)OTL(B14[24].8);
